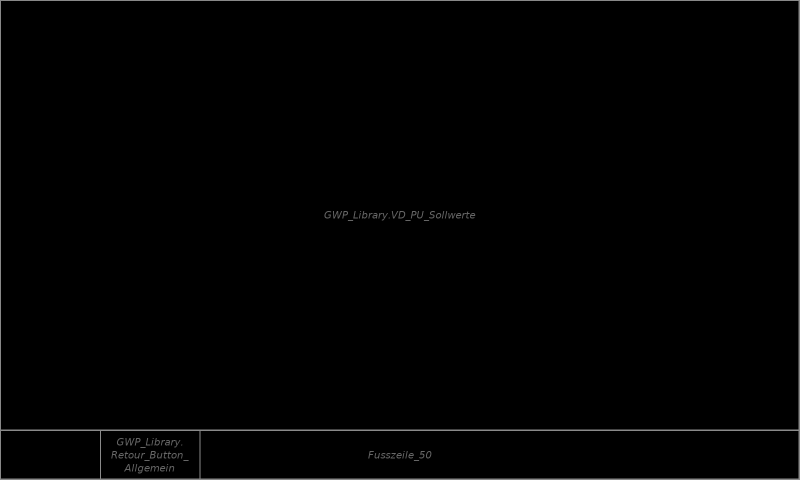
VISUALIZATION VD_PU_Sollwerte  // 800x480
    Frame (0,0 800x430)
        shows GWP_Library.VD_PU_Sollwerte(FB_VD := Main.VD_0)
    Frame (0,430 800x50)
        shows Fusszeile_50()
    Frame (100,430 100x50)
        shows GWP_Library.Retour_Button_Allgemein()
END_VISUALIZATION

(* stored: Version 1.1.0.1, ProductVersion 3.1.4022.6
   Visu VD_PU_Sollwerte: Id {161aea2f-cb5b-45ec-af75-274a1e20e8bc} *)
